(* IEC 61131-3 sources: myrepository/src, 5 files *)

(* ---- Average.st ---- *)
NAMESPACE SIMATIC.AX
    FUNCTION Average:REAL
        VAR_INPUT
            in1:REAL;
            in2:REAL;
        END_VAR
            Average:=(in1+in2)/2;
   END_FUNCTION
END_NAMESPACE

(* ---- cTankUnit.st ---- *)
USING Siemens.AxTest.Fluidhandling;
NAMESPACE Siemens.AxTest.Fluidhandling
Class public cTankUnit
    VAR PUBLIC
        cycleCount: INT;
        tank: cTank;
    END_VAR

    Method public mTankUnit
        VAR_INPUT
            cmdFill:bool;
            cmdEmptying : BOOL; // Outlet valve is open
            cmdFlush : BOOL; // Inlet and outlet valve is open
        END_VAR
        VAR_OUTPUT
            ctrlOpenInletValve:Bool;
            ctrlOpenOutletValve:Bool;
        END_VAR
    //instTank(cmdFill:=btnFill,cmdEmptying:=btnEmpty,cmdFlush:=btnFlush,inletValve:=inletValve,outletValve:=outletValve);//Valve作为INOUT
    tank.mTank(cmdFill:=cmdFill,cmdEmptying:=cmdEmptying,cmdFlush:=cmdFlush,ctrlOpenInletValve=>ctrlOpenInletValve,ctrlOpenOutletValve=>ctrlOpenOutletValve);
    //ctrlOpenInletValve:=inletValve.ctrlOpen;
    //ctrlOpenOutletValve:=outletValve.ctrlOpen;
    cycleCount := cycleCount + 1;
    END_METHOD
END_Class
END_NAMESPACE

NAMESPACE Siemen.AxTest.Fluidhandling
Function_Block UnitControl
    VAR
        unit:cTankUnit;
    END_VAR
    VAR_INPUT
        cmdFill : BOOL; // Inlet valve is open
        cmdEmptying : BOOL; // Outlet valve is open
        cmdFlush : BOOL; // Inlet and outlet valve is open
        //volume : LREAL;
    END_VAR
    VAR_OUTPUT
        ctrlOpenInletValve:Bool;
        ctrlOpenOutletValve:Bool;
    END_VAR
    unit.mTankUnit(cmdFill:=cmdFill,cmdEmptying:=cmdEmptying,cmdFlush:=cmdEmptying,ctrlOpenInletValve=>ctrlOpenInletValve,ctrlOpenOutletValve=>ctrlOpenOutletValve);
END_Function_Block
END_NAMESPACE

(* ---- Tank.st ---- *)
NAMESPACE Siemens.AxTest.Fluidhandling

    Class public cTank

        // VAR_IN_OUT
        //     inletValve : Valve;
        //     outletValve : Valve;
        // END_VAR

        VAR PUBLIC
            inletValve : REF_TO cValve;
            outletValve : REF_TO cValve;
        END_VAR
        method public mTank
            VAR_INPUT
                cmdFill : BOOL; // Inlet valve is open
                cmdEmptying : BOOL; // Outlet valve is open
                cmdFlush : BOOL; // Inlet and outlet valve is open
                //volume : LREAL;
            END_VAR
            VAR_OUTPUT
                ctrlOpenInletValve:Bool;
                ctrlOpenOutletValve:Bool;
            END_VAR
            VAR_TEMP
                tmpCmdInletOpen:bool;
                tmpCmdOutletOpen:bool;
            END_VAR
        IF (cmdFill XOR cmdEmptying XOR cmdFlush) THEN // check, if just one command is selected
            IF (cmdFill) THEN
                tmpCmdInletOpen := TRUE;
                tmpCmdOutletOpen := FALSE;
            ELSIF (cmdEmptying) THEN
                tmpCmdInletOpen := FALSE;
                tmpCmdOutletOpen := TRUE;
            ELSIF (cmdFlush) THEN
                tmpCmdInletOpen:= TRUE;
                tmpCmdOutletOpen := TRUE;
            END_IF;
        ELSE
            tmpCmdInletOpen:= FALSE;
            tmpCmdOutletOpen := FALSE;
        END_IF;
        ;
        inletValve^.mValve(cmdOpen:=tmpCmdInletOpen,ctrlOpen=>ctrlOpenInletValve);
        outletValve^.mValve(cmdOpen:=tmpCmdOutletOpen,ctrlOpen=>ctrlOpenOutletValve);
    end_method
    END_Class
END_NAMESPACE

(* ---- Valve.st ---- *)
using System.Timer;
NAMESPACE Siemens.AxTest.Fluidhandling
    Class PUBLIC cValve

        VAR PROTECTED
            cmdOpenOnDelay: OnDelay;
        END_VAR
        Method public mValve
            VAR_INPUT
                cmdOpen : BOOL;
            END_VAR
            VAR_OUTPUT
                ctrlOpen : BOOL;
                isOpen : BOOL;
                isClosed : BOOL;
            END_VAR
        cmdOpenOnDelay(signal:=cmdOpen,duration:=LT#2s);
        IF (cmdOpenOnDelay.OUTPUT) THEN

            isOpen := TRUE;
            isClosed := FALSE;
            ctrlOpen := TRUE;
        ELSE
            isOpen := FALSE;
            isClosed := TRUE;
            ctrlOpen := FALSE;
        END_IF;
    END_Method
    END_Class
END_NAMESPACE

(* ---- configuration.st ---- *)
using siemens.AxTest.Fluidhandling;
using System.Timer;
CONFIGURATION MyConfiguration
    TASK Main(Priority := 1);
    PROGRAM P1 WITH Main: MainProgramTank;

    VAR_GLOBAL
        //cmdOpenOndelay: OnDelay;

    END_VAR
    VAR_GLOBAL
        btnFill AT %I20.0:BOOL;
        btnEmpty AT %I20.1:BOOL;
        btnFlush AT %I20.2:Bool;
        ctrlOpenInletValve AT %Q20.0:Bool;
        ctrlOpenOutletValve AT %Q20.1:Bool;
        //actualVolume AT %MD20: REAL;
        inletValve:cValve;
        outletValve:cValve;
        tank:cTank := (inletValve:= REF(inletValve),outletValve:= REF(outletValve));
        //instUnitTank:  UnitControl;
    END_VAR
    VAR_GLOBAL
        dataArray:array[0..32767] of REAL;
        cycleCount:int;
    END_VAR
END_CONFIGURATION
PROGRAM MainProgramTank

    VAR_EXTERNAL
        // Inlet valve
        btnFill :BOOL;
        btnEmpty:BOOL;
        btnFlush:bool;
        ctrlOpenInletValve : BOOL;
        ctrlOpenOutletValve : BOOL;
        inletValve : cValve;
        outletValve:cValve;
        //instUnitTank : UnitControl;
        cycleCount : INT;
        tank: cTank;
    END_VAR

    VAR_TEMP
        //result : LREAL;
    END_VAR
    //cTank.inletValve:=REF(inletValve);
    //instTank(cmdFill:=btnFill,cmdEmptying:=btnEmpty,cmdFlush:=btnFlush,inletValve:=inletValve,outletValve:=outletValve);//Valve作为INOUT
    tank.mTank(cmdFill:=btnFill,cmdEmptying:=btnEmpty,cmdFlush:=btnFlush,ctrlOpenInletValve=>ctrlOpenInletValve,ctrlOpenOutletValve=>ctrlOpenOutletValve);
    //ctrlOpenInletValve:=inletValve.ctrlOpen;
    //ctrlOpenOutletValve:=outletValve.ctrlOpen;
    cycleCount := cycleCount + 1;
END_PROGRAM
